# EPICS autosave request: iocBoot/iocTomoScan_BEATS_FLIR_ACS_Step/auto_settings.req
file "tomoScan_settings.req", P=$(P), R=$(R)
file "tomoScan_BEATS_FLIR_ACS_Step_settings.req", P=$(P), R=$(R)
